FUNCTION_BLOCK DeserializationErrorFactory_TestSuite EXTENDS TcUnit.FB_TestSuite

TestCreateICustomDeserializationFailedError();
TestCreateIncorrectKeyTypeError();
TestCreateIncorrectTypeError();
TestCreateMissingKeyError();
TestCreateInvalidKeyError();

METHOD PUBLIC TestCreateICustomDeserializationFailedError
VAR
	error : CustomDeserializationFailedError('testMessage');
	factory : DeserializationErrorFactory;
	newError : I_Error;
END_VAR
TEST('TestCreateICustomDeserializationFailedError');

newError := factory.CreateCustomDeserializationFailedError('testMessage');

AssertTrue(
	Condition := newError.IsSameAs(error),
	Message := 'Did not produce the correct error type'
);

AssertEquals_String(
	Actual := newError.Message,
	Expected := error.Message,
	Message := 'Did not produce error with correct message'
);

newError.Dispose();

TEST_FINISHED();
END_METHOD

METHOD PUBLIC TestCreateIncorrectKeyTypeError
VAR
	error : IncorrectKeyTypeDeserializationError('testType', 'testKey');
	factory : DeserializationErrorFactory;
	newError : I_Error;
END_VAR
TEST('TestCreateIncorrectKeyTypeError');

newError := factory.CreateIncorrectKeyTypeError('testType','testKey');

AssertTrue(
	Condition := newError.IsSameAs(error),
	Message := 'Did not produce the correct error type'
);

AssertEquals_String(
	Actual := newError.Message,
	Expected := error.Message,
	Message := 'Did not produce error with correct message'
);

newError.Dispose();

TEST_FINISHED();
END_METHOD

METHOD PUBLIC TestCreateIncorrectTypeError
VAR
	error : IncorrectTypeDeserializationError('testType');
	factory : DeserializationErrorFactory;
	newError : I_Error;
END_VAR
TEST('TestCreateIncorrectTypeError');

newError := factory.CreateIncorrectTypeError('testType');

AssertTrue(
	Condition := newError.IsSameAs(error),
	Message := 'Did not produce the correct error type'
);

AssertEquals_String(
	Actual := newError.Message,
	Expected := error.Message,
	Message := 'Did not produce error with correct message'
);

newError.Dispose();

TEST_FINISHED();
END_METHOD

METHOD PUBLIC TestCreateInvalidKeyError
VAR
	error : InvalidKeyDeserializationError;
	factory : DeserializationErrorFactory;
	newError : I_Error;
END_VAR
TEST('TestCreateInvalidKeyError');

newError := factory.CreateInvalidKeyError();

AssertTrue(
	Condition := newError.IsSameAs(error),
	Message := 'Did not produce the correct error type'
);

AssertEquals_String(
	Actual := newError.Message,
	Expected := error.Message,
	Message := 'Did not produce error with correct message'
);

newError.Dispose();

TEST_FINISHED();
END_METHOD

METHOD PUBLIC TestCreateMissingKeyError
VAR
	error : MissingKeyDeserializationError('testKey');
	factory : DeserializationErrorFactory;
	newError : I_Error;
END_VAR
TEST('TestCreateMissingKeyError');

newError := factory.CreateMissingKeyError('testKey');

AssertTrue(
	Condition := newError.IsSameAs(error),
	Message := 'Did not produce the correct error type'
);

AssertEquals_String(
	Actual := newError.Message,
	Expected := error.Message,
	Message := 'Did not produce error with correct message'
);

newError.Dispose();

TEST_FINISHED();
END_METHOD

END_FUNCTION_BLOCK

(* stored: Version 1.1.0.1, ProductVersion 3.1.4024.12
   POU DeserializationErrorFactory_TestSuite: Id {3a25a940-1ef8-43b8-b103-fb414a2e3917}, SpecialFunc None
   Method TestCreateICustomDeserializationFailedError: Id {90e78d9a-f3f0-0dcc-24d7-05d854643abd}
   Method TestCreateIncorrectKeyTypeError: Id {eb81788b-0459-4a9c-9612-f2127bd2a320}
   Method TestCreateIncorrectTypeError: Id {587ace42-f928-4dd0-829f-038cc7883cf2}
   Method TestCreateInvalidKeyError: Id {51b97663-9b37-4a86-a55f-1f30062b9e9d}
   Method TestCreateMissingKeyError: Id {8e02c308-a62a-4de8-97ca-ac3c5aa17c6b} *)
